FUNCTION_BLOCK PUBLIC EventMsgParams
VAR_INPUT
	
END_VAR
VAR_OUTPUT
END_VAR
VAR
	CfgEvent                : TcEvent;
    fbEvent                 : ADSLOGEVENT;
    bSetEvent               : BOOL;(* Rising edge sets event *)
    eventData               : ST_EventData;
    TcEventDataFormatString : STRING    := '%f%d';
	bInitialize : BOOL := TRUE;
END_VAR

IF (bInitialize) THEN
	CfgEvent.Class := TCEVENTCLASS_ALARM;
	CfgEvent.Prio := 2;
	CfgEvent.Id := 1;
	CfgEvent.SourceId := 17001;
	CfgEvent.bQuitRequired := FALSE;//TRUE;
	CfgEvent.DataFormatStrAddress := ADR(TcEventDataFormatString);
	CfgEvent.Flags := TCEVENTFLAG_LOG OR TCEVENTFLAG_SRCID OR TCEVENTFLAG_AUTOFMTALL;
	CfgEvent.StreamType := TCEVENTSTREAM_SIMPLE;
	CfgEvent.ProgId :='TcEventFormatter.TcXMLFormatter' ;	
	eventData.rVal     := 0.00;
	eventData.iVal    := 0;
	bInitialize:= FALSE;	
END_IF

fbEvent(Event:=FALSE);

METHOD PUBLIC SendEventMsgParams : BOOL
VAR_INPUT
	MsgClass :		UDINT;
	EventID :		UDINT;
	SourceID : 		UDINT;
	RealVal: 		LREAL;
	IntVal :  		UDINT;
END_VAR
CfgEvent.Class := MsgClass;
CfgEvent.Id := EventID;
CfgEvent.SourceId := SourceID;
eventData.rVal := RealVal;
eventData.iVal := IntVal;
fbEvent( NETID:= '',
        PORT:= 110,
        Event:=TRUE,
        EventConfigData:= CfgEvent,
        EventDataAddress := ADR(eventData) ,
    	EventDataLength := SIZEOF(eventData),
        TMOUT:= T#3S);
END_METHOD

END_FUNCTION_BLOCK

(* stored: Version 1.1.0.1, ProductVersion 3.1.4020.12
   POU EventMsgParams: Id {eb16ca0e-af54-4630-b5ca-b77de0962b32}, SpecialFunc None
   Method SendEventMsgParams: Id {52991bbc-184b-40c6-bfc9-bb715b8eaabc} *)
